# EPICS autosave request: optics/opticsApp/Db/MLLV_soft_settings.req
$(P)$(Q)zLen
$(P)$(Q)yLen
file basic_motor_settings.req P=$(P),Q=$(Q),M=$(Q)th
file basic_motor_settings.req P=$(P),Q=$(Q),M=$(Q)z
file basic_motor_settings.req P=$(P),Q=$(Q),M=$(Q)y
file basic_motor_settings.req P=$(P),Q=$(Q),M=$(Q)chi
file basic_motor_settings.req P=$(P),Q=$(Q),M=$(Q)x
